INTERFACE ITF_ControlElement_HMI_1 EXTENDS ITF_BaseControlElement_HMI

METHOD LinkControlElementData : BOOL
VAR_INPUT
	stData				: REFERENCE TO ST_ControlElement_HMI_Link;
END_VAR
END_METHOD

END_INTERFACE

(* stored: Version 1.1.0.1, ProductVersion 3.1.4024.15
   Itf ITF_ControlElement_HMI_1: Id {51dbf68b-e225-45ea-a15c-b9da8b6506cd}
   Method LinkControlElementData: Id {c304068a-6076-4f72-a703-2420149dbf31} *)
